(* LS Electric XG5000 project: 3_MY_Auto_Start_Delta *)
(* PLC LSPLC *)

PROGRAM NewProgram (* task: Scan Program *)
VAR
    INST : TON;
    MC_C : BOOL;
    MC_D AT %QX0.0.1 : BOOL;
    MC_S AT %QX0.0.2 : BOOL;
    PBS_Off AT %IX0.0.1 : BOOL;
    PBS_ON AT %IX0.0.0 : BOOL;
END_VAR

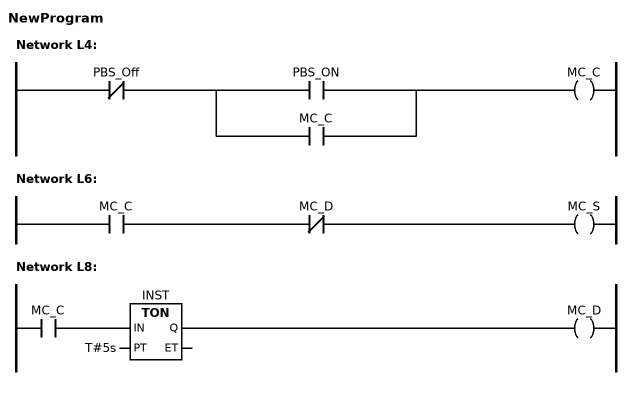
(* Rung L4 *)
MC_C := NOT PBS_Off AND (PBS_ON OR MC_C);
(* Rung L6 *)
MC_S := MC_C AND NOT MC_D;
(* Rung L8 *)
INST(IN := MC_C, PT := T#5s);
MC_D := INST.Q;
END_PROGRAM